// TIA Portal V17 export
// export: Created 2024-06-14T09:53:02.5761361Z, ExportSetting WithDefaults, DisplayName Totally Integrated Automation Portal, DisplayVersion V17, DisplayName TIA Portal Openness, DisplayVersion V17, DisplayName TIA Portal Version Control Interface, DisplayVersion V17, DisplayName Simotion SCOUT TIA, DisplayVersion 5.4.3.0, DisplayName SINAMICS Startdrive Advanced, DisplayVersion V17 SP1 Update 1, DisplayName SINAMICS Startdrive G110M, G120, G120C, G120D, G120P, G115D, DisplayVersion V17 SP1 Update 1, DisplayName SINAMICS Startdrive G130, G150, S120, S150, SINAMICS MV, S210, DisplayVersion V17 SP1 Update 1, DisplayName STEP 7 Professional, DisplayVersion V17, DisplayName STEP 7 Safety, DisplayVersion V17, DisplayName WinCC Professional, DisplayVersion V17
DATA_BLOCK "CylinderSetup_DB"   // DB28
{ S7_Optimized_Access := 'FALSE' }
VERSION : 0.1
// stored: AutoNumber true, DBAccessibleFromOPCUA true, IsOnlyStoredInLoadMemory false, IsWriteProtectedInAS false
   VAR
      Array_S1 { S7_SetPoint := 'True'} : Array[1..50] of "uCylinderData";
      Array_S2 { S7_SetPoint := 'True'} : Array[1..50] of "uCylinderData";
      Array_S3 { S7_SetPoint := 'True'} : Array[1..50] of "uCylinderData";
      Array_S4 { S7_SetPoint := 'True'} : Array[1..50] of "uCylinderData";
      Array_S5 { S7_SetPoint := 'True'} : Array[1..50] of "uCylinderData";
      Array_S6 { S7_SetPoint := 'True'} : Array[1..50] of "uCylinderData";
      Array_S7 { S7_SetPoint := 'True'} : Array[1..50] of "uCylinderData";
      Array_S8 { S7_SetPoint := 'True'} : Array[1..50] of "uCylinderData";
      Array_S9 { S7_SetPoint := 'True'} : Array[1..50] of "uCylinderData";
      Array_S10 { S7_SetPoint := 'True'} : Array[1..50] of "uCylinderData";
      Array_S11 { S7_SetPoint := 'True'} : Array[1..50] of "uCylinderData";
      Array_S1_Data : Struct
         Length : Int;
      END_STRUCT;
      Array_S2_Data : Struct
         Length : Int;
      END_STRUCT;
      Array_S3_Data : Struct
         Length : Int;
      END_STRUCT;
      Array_S4_Data : Struct
         Length : Int;
         Array_S2_Data : Struct
            Length : Int;
         END_STRUCT;
      END_STRUCT;
      Array_S5_Data_1 : Struct
         Length : Int;
         Array_S3_Data : Struct
            Length : Int;
         END_STRUCT;
      END_STRUCT;
      "No.OfItems TO S2" : Int := 0;
      Array_R1 { S7_SetPoint := 'True'} : Array[1..50] of "uCylinderData";
      "No.OfItems TO S3" : Int := 0;
      "No.OfItems TO S4" : Int := 0;
      "No.OfItems TO S5" : Int := 0;
      "No.OfItems TO S6" : Int := 1;
      "No.OfItems TO S7" : Int;
      "No.OfItems TO S8" : Int;
      Array_R1_Data : Struct
         Length : Int;
      END_STRUCT;
      Tare_Entry : Real;
   END_VAR
BEGIN
   Array_S6[1].rCylinderID := 0;
   Array_S6[1].rNet_weight := 0.0;
   Array_S6[1].rTareWeight := 0.0;
   Array_S6[1].rGross_Weight := 0.0;
   Array_S6[1].iCylinderType := 0;
END_DATA_BLOCK
